// Implicitly generated code : DO NOT EDIT
FUNCTION CheckDivDInt : DINT
VAR_INPUT
    divisor : DINT;
END_VAR

// Implicitly generated code : Only an Implementation suggestion
{noflow}
IF divisor = 0 THEN
    CheckDivDInt := 1;
ELSE
    CheckDivDInt := divisor;
END_IF;
{flow}

END_FUNCTION

(* stored: Version 1.1.0.1
   POU CheckDivDInt: Id {ce67f877-aa83-0475-2148-bd8a848aabd0}, SpecialFunc CheckDivInt32 *)
